TYPE SignalBlockBase :
STRUCT
END_STRUCT
END_TYPE

(* stored: Version 1.1.0.1, ProductVersion 3.1.4020.12
   DUT SignalBlockBase: Id {bdbdac30-612d-430e-bbcf-43f1cafaa021} *)
